TYPE PID_Parameter_Strukt :
STRUCT
	Kp :		REAL;
	Ti :		REAL;
	Td :		REAL;
	N :			REAL;
	ARW :		REAL;
	umin :		REAL;
	umax :		REAL;
END_STRUCT
END_TYPE

(* stored: Version 1.1.0.1, ProductVersion 3.1.4024.13
   DUT PID_Parameter_Strukt: Id {00266e82-5d55-4001-a92e-a7de3af1a787} *)
